PROGRAM SimulationMAIN
VAR
	cylinder_stub:	Cylinder;
	io: cylinder2IO;
	push_stroke_time: REAL := 1.8;
	pull_stroke_time: REAL := 1.5;
	chattering_time: REAL := 0.5;
END_VAR

cylinder_stub.push_time := REAL_TO_TIME(push_stroke_time * 1000);
cylinder_stub.pull_time := REAL_TO_TIME(pull_stroke_time * 1000);
cylinder_stub.chattering_time := REAL_TO_TIME(chattering_time * 1000);

cylinder_stub(io:= io);

END_PROGRAM

(* stored: Version 1.1.0.1, ProductVersion 3.1.4024.12
   POU SimulationMAIN: Id {6768b7e2-d7cc-451c-be66-683fbc082fff}, SpecialFunc None *)
